PROGRAM prgLynus
VAR
	fbRW1		: FB_ReadWrite_V2;
END_VAR

fbRW1(
	eUploadType:= eSelectDataUploadType.e_Change_Intervall5min , 
	bBusy=> , 
	bError=> , 
	udiErrorCodeOut=> , 
	eErrorReadWrite_Out=> );

END_PROGRAM

(* stored: Version 1.1.0.1, ProductVersion 3.1.4024.11
   POU prgLynus: Id {32763d1c-6f6f-414b-994c-074000e28f24}, SpecialFunc None *)
